# EPICS autosave request: iocBoot/ioc13raman/auto_positions.req
file "CARS_motor_positions.req",         P=13Raman:, M=m1
file "CARS_motor_positions.req",         P=13Raman:, M=m2
file "CARS_motor_positions.req",         P=13Raman:, M=m3
~
